PROGRAM driveTestCall
VAR

	//instances for each motion of the drive
	driveMotion1: FB_DriveMotion;
	driveMotion2: FB_DriveMotion;
	driveMotion3: FB_DriveMotion;
	//instance for the call inside the PLC
	driveMotionCall: FB_DriveInterface;
END_VAR

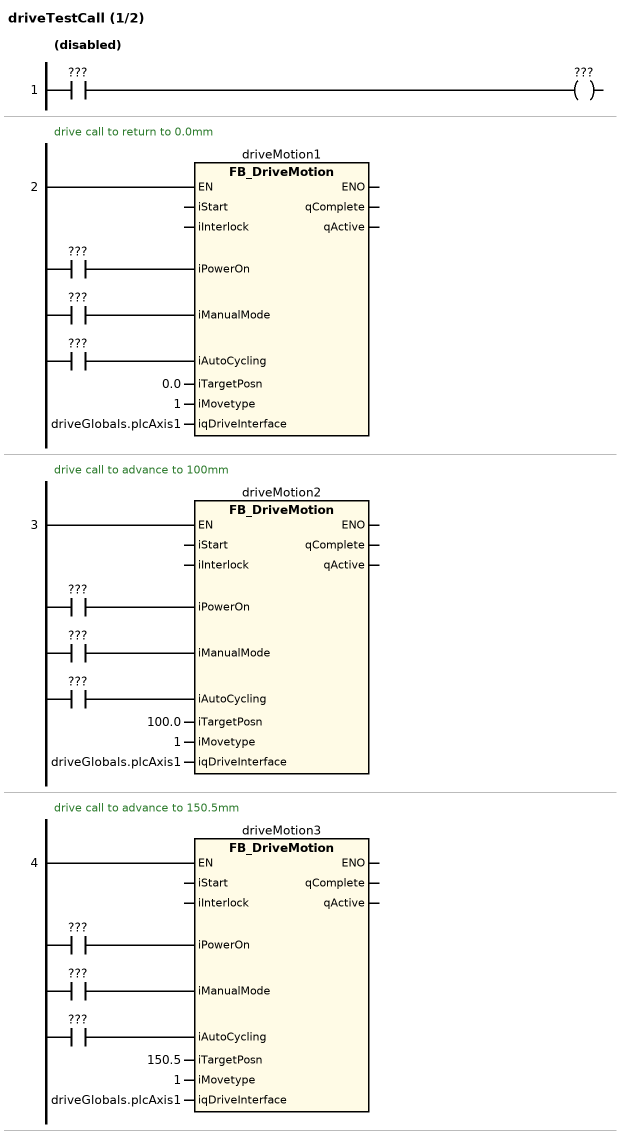
// NETWORK 1 (disabled)
// ??? := ???;

// NETWORK 2
// drive call to return to 0.0mm
driveMotion1(iTargetPosn := 0.0, iMovetype := 1, iqDriveInterface := driveGlobals.plcAxis1); // FB_DriveMotion

// NETWORK 3
// drive call to advance to 100mm
driveMotion2(iTargetPosn := 100.0, iMovetype := 1, iqDriveInterface := driveGlobals.plcAxis1); // FB_DriveMotion

// NETWORK 4
// drive call to advance to 150.5mm
driveMotion3(iTargetPosn := 150.5, iMovetype := 1, iqDriveInterface := driveGlobals.plcAxis1); // FB_DriveMotion

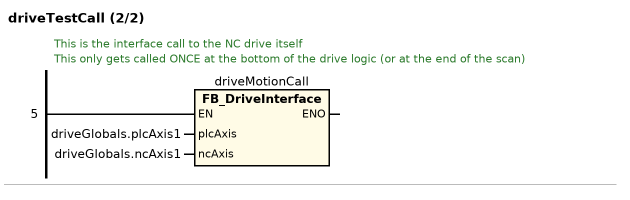
// NETWORK 5
// This is the interface call to the NC drive itself
// This only gets called ONCE at the bottom of the drive logic (or at the end of the scan)
driveMotionCall(plcAxis := driveGlobals.plcAxis1, ncAxis := driveGlobals.ncAxis1); // FB_DriveInterface

END_PROGRAM

(* stored: Version 1.1.0.1, ProductVersion 3.1.4024.12
   POU driveTestCall: Id {d6a677ea-9647-4d36-8e56-9ba6621c13d7}, SpecialFunc None *)
